(* IEC 61131-3 sources: 2026_Projet_YGO_ExcavatriceDragage/DOC/WFLOW/AUDITS, 1 file *)

(* ---- FB_Cycle_proposal.st ---- *)
(* ═══════════════════════════════════════════════════════════════
   🔄 FB_Cycle — Séquenceur du Cycle Automatique (Grafcet de dragage)
   ───────────────────────────────────────────────────────────────
   📄 Doc : DOC/AF/AF_Partie-04_Mode_SemiAuto_Sequenceur_v2.0.md
            DOC/WFLOW/AUDITS/DESIGN_SEMI_AUTO_CYCLE_v0.1.md
   🔌 Conforme au contrat FB standard (Partie3 §1bis) + §11bis R1-R9.
   🧩 Deux instances : instCycleMaintenance (MAINT_N1/N2) et
      instCycleSemiAuto (SEMI_AUTO) — gating sorties par mode.
   🕹️ Homme-mort (D2) : appui = autorisation 3 s ; mouvement continue
      sans appui ; arrêt au centre du manche (CycleMotionPermit).
   ⏱️ Tempo max d'étape : lancée SEULEMENT si pilotage joystick actif.
   🧊 CycleStepAtError : étape spécifique mémorisée avant STABILIZING (R9).
   🏁 Début de graphe : à la TRÉMIE, treuils en position HAUTE — rebouclage sur X0.
   ═══════════════════════════════════════════════════════════════ *)

FUNCTION_BLOCK PUBLIC FB_Cycle
VAR_INPUT
    Enable                  : BOOL;         // Activation générale du séquenceur
    Reset                   : BOOL;         // Acquittement défaut (front)
    PowerContactorEngaged   : BOOL;         // Chaîne de sécurité OK
    Mode                    : E_Mode;       // Mode arbitré (SEMI_AUTO pour l'instance cycle)
    CycleMotionPermit       : BOOL;         // 🕹️ Manche défléchi (non centré) — D2
    DeadmanArmed            : BOOL;         // 🔫 Appui homme-mort (fenêtre 3 s)
    HeartbeatIhmOk          : BOOL;         // 💓 IHM↔PLC valide

    // Commandes opérateur
    StartCycle              : BOOL;         // Demande lancement / reprise (IHM)
    AbortCycle              : BOOL;         // Demande abandon (IHM) — pas de Pause (D3)

    // Cibles et paramètres (réutilise config maintenance — Q4)
    SelTarget               : INT;          // 🎯 Cible sélectionnée (GVL_IHM.TranslationM3.Cmd.SelTarget) : 1=Trémie, 2=P2, 3=P1, 4=Maintenance
    SetDepthM               : REAL;         // Profondeur de consigne (négative)
    SetOffsetM              : REAL;         // Écart de fermeture benne cible

    // Feedbacks physique & matériel
    KoboldContactFond       : BOOL;         // Retour dédié Kobold : TRUE = contact fond
    LimitLegalReached       : BOOL;         // Limite légale atteinte (descente interdite)
    LimitLegalDepthM        : REAL;         // Profondeur légale minimale autorisée
    WinchSyncError          : BOOL;         // Désynchronisme bloquant M1/M2
    WinchSyncDeltaM         : REAL;         // Écart codeurs M1/M2 pour diagnostic
    M1_CablePosM            : REAL;         // Position câble treuil M1 (recalée)
    M2_CablePosM            : REAL;         // Position câble treuil M2 (recalée)
    M1_MeasuredSpeedMps     : REAL;         // Vitesse linéaire mesurée M1 (m/s)
    M2_MeasuredSpeedMps     : REAL;         // Vitesse linéaire mesurée M2 (m/s)
    SpeedMismatchThresholdMps : REAL;       // Seuil écart vitesse ; 0 = contrôle désactivé
    SpeedMismatchTimeout    : TIME;         // Durée de confirmation ; 0 = contrôle désactivé
    CableLimitM1AscentM     : REAL;         // Limite haute d'exploitation M1

    // Feedbacks Translation M3
    Translation_At_P1           : BOOL;     // Capteur position P1 (arrêt travail)
    Translation_At_Tremie       : BOOL;     // Capteur fin de course trémie
    Translation_At_Maintenance : BOOL;     // Capteur fin de course maintenance
    Translation_Busy            : BOOL;     // Mouvement translation en cours
    Translation_Done            : BOOL;     // Cible translation atteinte

    // Feedbacks Benne
    Benne_Busy              : BOOL;         // Mouvement mâchoires benne en cours
    Benne_Done              : BOOL;         // Mouvement ouverture/fermeture terminé
    Benne_IsOpen            : BOOL;         // Benne mécaniquement ouvert mémorisé
    Benne_IsClosed          : BOOL;         // Benne mécaniquement fermé mémorisé
    Benne_IsRoughlyClosed   : BOOL;         // 🆕 Benne « à peu près fermée » (tolérance matière)

    // 🆕 Référencement (X1_HOMING)
    HomedM1                 : BOOL;         // Codeur M1 référencé
    HomedM2                 : BOOL;         // Codeur M2 référencé
    TopPositionSensor       : BOOL;         // Capteur position haute (référencement)
    HomingRequest           : BOOL;         // Demande de référencement (front)
END_VAR
VAR_OUTPUT
    Ready                   : BOOL;         // Séquenceur disponible
    Busy                    : BOOL;         // Cycle automatique actif
    Done                    : BOOL;         // Cycle automatique complété
    Error                   : BOOL;         // Défaut cycle
    ErrorId                 : WORD;         // bit0: timeout/limite, bit1: désynchronisme, bit2: cible invalide, bit3: stabilisation impossible, bit4: écart vitesse, bit5: perte heartbeat, bit6: tempo max étape
    SpeedMismatchMps        : REAL;         // Écart absolu vitesse M1/M2 (m/s)
    SpeedMismatchActive     : BOOL;         // Seuil vitesse dépassé sur le cycle courant
    SpeedMismatchConfirmed  : BOOL;         // Écart vitesse confirmé pendant SpeedMismatchTimeout

    // Commandes structurées (demandes de mouvement)
    WinchM1Cmd              : ST_WinchCmdDemand;        // Demande treuil M1
    WinchM2Cmd              : ST_WinchCmdDemand;        // Demande treuil M2
    TranslationCmd          : ST_TranslationCmdDemand;  // Demande translation M3
    BucketCmd               : ST_BucketCmdDemand;       // Demande benne

    // Métadonnées d'affichage IHM
    CycleStep               : E_CycleStep;  // Étape active du Grafcet
    CycleStateStr           : STRING(80);   // Libellé en clair de l'étape (Xn - texte)
    CycleStepAtError        : E_CycleStep;  // 🧊 Étape spécifique au moment du défaut (R9)
    SampleCount             : INT;          // 🆕 Compteur de prélèvements (RETAIN, Q3bis)
END_VAR
VAR
    ResetEdge               : R_TRIG;
    StartEdge               : R_TRIG;
    AbortEdge               : R_TRIG;
    ErrorEdge               : R_TRIG;       // 🧊 Capture CycleStepAtError avant bascule (R9)

    // Séquencement
    State                   : E_CycleStep := E_CycleStep.X0_PREPARATION;
    SavedState              : E_CycleStep := E_CycleStep.X0_PREPARATION;

    // Mémorisations et Timers
    TouchPositionM          : REAL;         // Position M1 mémorisée lors du contact fond
    RaiseTargetM            : REAL;         // Profondeur de remontée mémorisée
    DrainingTimer           : TON;          // Temporisateur de vidage (égouttage)
    StabilizationTimer      : TON;          // Temporisation maximale de remontée lente
    SpeedMismatchTimer      : TON;          // Confirmation temporelle écart de vitesse
    StepMaxTimer            : TON;          // 🆕 Tempo max d'étape (R5) — lancée si pilotage
    SelectedWorkTarget      : INT;          // Cible de travail mémorisée (1=Trémie, 3=P1, 4=Maintenance)

    // Paramètres internes
    CtrlAscentDistM         : REAL := 2.0;      // Distance de remontée lente de contrôle
    CtrlAscentToleranceM    : REAL := 0.25;     // Écart maximal admis entre les deux codeurs
    CtrlAscentTimeout       : TIME := T#30s;    // Temps max pour atteindre la zone de stabilisation
    DrainingTime            : TIME := T#5s;     // Temps d'égouttage par défaut
    StepMaxTimeout          : TIME := T#60s;   // 🆕 Tempo max d'étape (à valider, Q4)
END_VAR

// === IMPLEMENTATION ===

{region "Gate securite"}
// 🛑 1. GATES DE SÉCURITÉ ET BLOCAGE (R8)
IF NOT Enable OR NOT PowerContactorEngaged THEN
    WinchM1Cmd.StartStop   := FALSE;
    WinchM1Cmd.Direction   := 0;
    WinchM1Cmd.SpeedPct    := 0.0;

    WinchM2Cmd.StartStop   := FALSE;
    WinchM2Cmd.Direction   := 0;
    WinchM2Cmd.SpeedPct    := 0.0;

    TranslationCmd.Start   := FALSE;
    TranslationCmd.Target  := 0;

    BucketCmd.Open         := FALSE;
    BucketCmd.Close        := FALSE;
    BucketCmd.KoboldContactorCmd := FALSE;

    State                := E_CycleStep.X0_PREPARATION;   // retour à la PREMIÈRE étape (R8)
    CycleStep            := E_CycleStep.X0_PREPARATION;
    CycleStateStr        := 'X0 - Désactivé : sécurité absente ou auto désactivé';
    Ready                := FALSE;
    Busy                 := FALSE;
    Done                 := FALSE;
    RETURN;
END_IF;
{endregion}

{region "Preparation surveillance et commandes cycle"}
Ready := TRUE;
ResetEdge(CLK := Reset);
StartEdge(CLK := StartCycle);
AbortEdge(CLK := AbortCycle);
ErrorEdge(CLK := Error);

// 🧊 R9 — capture l'étape spécifique AVANT la bascule vers STABILIZING
IF ErrorEdge.Q THEN
    CycleStepAtError := State;
END_IF;

// ⏱️ T36 — surveillance indépendante de la remontée lente
StabilizationTimer(IN := (State = E_CycleStep.X7_CTRL_ASCENT), PT := CtrlAscentTimeout);

// 📏 T43 — comparaison vitesse réelle M1/M2
SpeedMismatchMps := ABS(M1_MeasuredSpeedMps - M2_MeasuredSpeedMps);
SpeedMismatchActive := (State = E_CycleStep.X7_CTRL_ASCENT)
                       AND CycleMotionPermit
                       AND (SpeedMismatchThresholdMps > 0.0)
                       AND (SpeedMismatchTimeout > T#0ms)
                       AND (SpeedMismatchMps > SpeedMismatchThresholdMps);
SpeedMismatchTimer(IN := SpeedMismatchActive, PT := SpeedMismatchTimeout);
SpeedMismatchConfirmed := SpeedMismatchTimer.Q;

// 🆕 Tempo max d'étape (R5) — lancée SEULEMENT si pilotage joystick actif (pas de défaut au repos)
StepMaxTimer(IN := CycleMotionPermit AND (State <> E_CycleStep.X0_PREPARATION)
                  AND (State <> E_CycleStep.X13_DONE_SYNC)
                  AND (State <> E_CycleStep.STABILIZING),
             PT := StepMaxTimeout);

IF ResetEdge.Q THEN
    Error := FALSE;
    ErrorId := 16#0000;
    SavedState := E_CycleStep.X0_PREPARATION;
    IF State = E_CycleStep.STABILIZING THEN
        State := E_CycleStep.X0_PREPARATION;
    END_IF;
END_IF;

// 💓 Perte IHM : repli mémorisé. La reconnexion seule ne relance jamais le cycle.
IF NOT HeartbeatIhmOk AND State <> E_CycleStep.STABILIZING THEN
    Error := TRUE;
    ErrorId := ErrorId OR 16#0020;
    State := E_CycleStep.STABILIZING;
END_IF;

// Défaut de synchronisme : arrêt sûr et acquittement obligatoire.
IF WinchSyncError AND State <> E_CycleStep.STABILIZING THEN
    Error := TRUE;
    ErrorId := ErrorId OR 16#0002;
    State := E_CycleStep.STABILIZING;
END_IF;

// 🛡️ T43 — écart de vitesse confirmé : arrêt du cycle et STABILIZING.
IF SpeedMismatchConfirmed AND State <> E_CycleStep.STABILIZING THEN
    Error := TRUE;
    ErrorId := ErrorId OR 16#0010;
    State := E_CycleStep.STABILIZING;
END_IF;

// 🆕 Tempo max d'étape dépassée (blocage probable) → défaut
IF StepMaxTimer.Q AND State <> E_CycleStep.STABILIZING THEN
    Error := TRUE;
    ErrorId := ErrorId OR 16#0040;
    State := E_CycleStep.STABILIZING;
END_IF;

// Gestion de l'Abandon (D3 — pas de Pause)
IF AbortEdge.Q THEN
    State := E_CycleStep.X0_PREPARATION;
END_IF;
{endregion}

{region "Machine etat cycle automatique"}
// 🔁 2. LOGIQUE DU SÉQUENCEUR (Machine d'état) — CASE sur enum unique (R1)
CASE State OF

    E_CycleStep.X0_PREPARATION:
        CycleStep := E_CycleStep.X0_PREPARATION;
        CycleStateStr := 'X0 - Vérification cohérence système';
        WinchM1Cmd.StartStop := FALSE; WinchM1Cmd.Direction := 0; WinchM1Cmd.SpeedPct := 0.0;
        WinchM2Cmd.StartStop := FALSE; WinchM2Cmd.Direction := 0; WinchM2Cmd.SpeedPct := 0.0;
        TranslationCmd.Start := FALSE; TranslationCmd.Target := 0;
        BucketCmd.Open := FALSE; BucketCmd.Close := FALSE; BucketCmd.KoboldContactorCmd := FALSE;
        Busy := FALSE; Done := FALSE;

        // Transition si système sain et réarmé (front reset ou démarrage)
        IF StartEdge.Q THEN
            State := E_CycleStep.X1_HOMING;
        END_IF;

    E_CycleStep.X1_HOMING:
        CycleStep := E_CycleStep.X1_HOMING;
        CycleStateStr := 'X1 - Référencement codeurs (vitesses lentes)';
        Busy := TRUE;

        // 🆕 Vitesses lentes pour chercher capteur top + référencement
        IF NOT HomedM1 OR NOT HomedM2 THEN
            WinchM1Cmd.StartStop := CycleMotionPermit;
            WinchM1Cmd.Direction := 1;   // montée lente vers capteur top
            WinchM1Cmd.SpeedPct := 10.0;
            WinchM2Cmd.StartStop := CycleMotionPermit;
            WinchM2Cmd.Direction := 1;
            WinchM2Cmd.SpeedPct := 10.0;
            IF HomingRequest THEN
                // déclenche le référencement (via FB_Encoder_Homing en aval)
                State := E_CycleStep.X2_WORK_POS_SELECT;
            END_IF;
        ELSE
            // déjà homé → passe vite
            State := E_CycleStep.X2_WORK_POS_SELECT;
        END_IF;

    E_CycleStep.X2_WORK_POS_SELECT:
        CycleStep := E_CycleStep.X2_WORK_POS_SELECT;
        CycleStateStr := 'X2 - Sélection position travail (P1)';
        Busy := TRUE;

        // 🆕 Destinations sélectionnables : Trémie(1), P1(3), Maintenance(4).
        // P2(2) n'est PAS une destination — capteur de passage en petite vitesse (PV).
        IF (SelTarget <> 1) AND (SelTarget <> 3) AND (SelTarget <> 4) THEN
            Error := TRUE;
            ErrorId := ErrorId OR 16#0004;
            State := E_CycleStep.STABILIZING;
        ELSE
            SelectedWorkTarget := SelTarget;
            TranslationCmd.Target := SelTarget;
            TranslationCmd.Start := CycleMotionPermit;
            // Arrivée à la cible (Trémie/P1/Maintenance) — capteurs PV/PVP2/P2 = ralentissement
            IF CycleMotionPermit AND (
                (SelTarget = 1 AND Translation_At_Tremie) OR
                (SelTarget = 3 AND Translation_At_P1) OR
                (SelTarget = 4 AND Translation_At_Maintenance)) THEN
                TranslationCmd.Start := FALSE;
                State := E_CycleStep.X3_OPEN_BUCKET;
            END_IF;
        END_IF;

    E_CycleStep.X3_OPEN_BUCKET:
        CycleStep := E_CycleStep.X3_OPEN_BUCKET;
        CycleStateStr := 'X3 - Ouverture benne';
        Busy := TRUE;

        // 🆕 Ouverture benne ; si déjà ouverte → passe vite
        IF Benne_IsOpen THEN
            State := E_CycleStep.X4_DESCEND_OPEN;
        ELSE
            BucketCmd.Open := CycleMotionPermit;
            IF CycleMotionPermit AND Benne_Done AND Benne_IsOpen THEN
                BucketCmd.Open := FALSE;
                State := E_CycleStep.X4_DESCEND_OPEN;
            END_IF;
        END_IF;

    E_CycleStep.X4_DESCEND_OPEN:
        CycleStep := E_CycleStep.X4_DESCEND_OPEN;
        CycleStateStr := 'X4 - Plongée benne ouverte (synchro)';

        // M1 et M2 descendent ensemble (synchro gérée en aval)
        WinchM1Cmd.StartStop := CycleMotionPermit;
        WinchM1Cmd.Direction := -1;
        WinchM1Cmd.SpeedPct  := 50.0;
        WinchM2Cmd.StartStop := CycleMotionPermit;
        WinchM2Cmd.Direction := -1;
        WinchM2Cmd.SpeedPct  := 50.0;
        BucketCmd.KoboldContactorCmd := TRUE;

        // Transition uniquement sur le retour dédié Kobold.
        IF CycleMotionPermit AND KoboldContactFond THEN
            WinchM1Cmd.StartStop := FALSE;
            WinchM2Cmd.StartStop := FALSE;
            BucketCmd.KoboldContactorCmd := FALSE;
            TouchPositionM := M1_CablePosM;
            IF LimitLegalDepthM < -0.01 THEN
                RaiseTargetM := MAX(TouchPositionM + 0.5, LimitLegalDepthM + 0.5);
            ELSE
                RaiseTargetM := TouchPositionM + 0.5;
            END_IF;
            State := E_CycleStep.X5_BOTTOM_CONFIRMED;
        ELSIF LimitLegalReached THEN
            Error := TRUE;
            ErrorId := ErrorId OR 16#0001;
            WinchM1Cmd.StartStop := FALSE;
            WinchM2Cmd.StartStop := FALSE;
            BucketCmd.KoboldContactorCmd := FALSE;
            State := E_CycleStep.STABILIZING;
        END_IF;

    E_CycleStep.X5_BOTTOM_CONFIRMED:
        CycleStep := E_CycleStep.X5_BOTTOM_CONFIRMED;
        CycleStateStr := 'X5 - Fond confirmé : remontée sécurisée';

        WinchM1Cmd.StartStop := CycleMotionPermit;
        WinchM1Cmd.Direction := 1;
        WinchM1Cmd.SpeedPct := 20.0;
        WinchM2Cmd.StartStop := CycleMotionPermit;
        WinchM2Cmd.Direction := 1;
        WinchM2Cmd.SpeedPct := 20.0;

        // Les deux treuils restent synchronisés jusqu'au-dessus de la limite légale.
        IF CycleMotionPermit AND (M1_CablePosM >= RaiseTargetM) AND (M2_CablePosM >= RaiseTargetM) THEN
            WinchM1Cmd.StartStop := FALSE;
            WinchM2Cmd.StartStop := FALSE;
            State := E_CycleStep.X6_CLOSE_BUCKET;
        END_IF;

    E_CycleStep.X6_CLOSE_BUCKET:
        CycleStep := E_CycleStep.X6_CLOSE_BUCKET;
        CycleStateStr := 'X6 - Fermeture benne (tolérance à peu près fermé)';

        WinchM1Cmd.StartStop := FALSE;
        BucketCmd.Close := TRUE;

        // 🆕 Tolérance : si benne « à peu près fermée » (matière/objet), on remonte et on contrôle
        IF CycleMotionPermit AND (Benne_Done AND (Benne_IsClosed OR Benne_IsRoughlyClosed)) THEN
            BucketCmd.Close := FALSE;
            State := E_CycleStep.X7_CTRL_ASCENT;
        END_IF;

    E_CycleStep.X7_CTRL_ASCENT:
        CycleStep := E_CycleStep.X7_CTRL_ASCENT;
        CycleStateStr := 'X7 - Remontée lente de contrôle';

        WinchM1Cmd.StartStop := CycleMotionPermit;
        WinchM1Cmd.Direction := 1;
        WinchM1Cmd.SpeedPct  := 20.0;
        WinchM2Cmd.StartStop := CycleMotionPermit;
        WinchM2Cmd.Direction := 1;
        WinchM2Cmd.SpeedPct  := 20.0;

        // Contrôle des deux codeurs
        IF WinchSyncError OR (ABS(M1_CablePosM - M2_CablePosM) > CtrlAscentToleranceM) THEN
            Error := TRUE;
            ErrorId := ErrorId OR 16#0008;
            State := E_CycleStep.STABILIZING;
        ELSIF CycleMotionPermit
           AND (M1_CablePosM >= (TouchPositionM + CtrlAscentDistM))
           AND (M2_CablePosM >= (TouchPositionM + CtrlAscentDistM))
           AND (ABS(M1_CablePosM - M2_CablePosM) <= CtrlAscentToleranceM) THEN
            State := E_CycleStep.X8_ASCENT_LOADED;
        ELSIF StabilizationTimer.Q THEN
            Error := TRUE;
            ErrorId := ErrorId OR 16#0008;
            State := E_CycleStep.STABILIZING;
        END_IF;

    E_CycleStep.X8_ASCENT_LOADED:
        CycleStep := E_CycleStep.X8_ASCENT_LOADED;
        CycleStateStr := 'X8 - Remontée en charge';

        WinchM1Cmd.StartStop := CycleMotionPermit;
        WinchM1Cmd.Direction := 1;
        WinchM1Cmd.SpeedPct  := 70.0;
        WinchM2Cmd.StartStop := CycleMotionPermit;
        WinchM2Cmd.Direction := 1;
        WinchM2Cmd.SpeedPct  := 70.0;

        // Transition alignée sur la limite haute d'exploitation
        IF CycleMotionPermit AND M1_CablePosM >= CableLimitM1AscentM THEN
            WinchM1Cmd.StartStop := FALSE;
            WinchM2Cmd.StartStop := FALSE;
            State := E_CycleStep.X9_DRAIN_PAUSE;
        END_IF;

    E_CycleStep.X9_DRAIN_PAUSE:
        CycleStep := E_CycleStep.X9_DRAIN_PAUSE;
        CycleStateStr := 'X9 - Égouttage du godet en cours';
        WinchM1Cmd.StartStop := FALSE;
        WinchM2Cmd.StartStop := FALSE;

        DrainingTimer(IN := TRUE, PT := DrainingTime);
        // 🆕 Temps écoulé affiché IHM (CycleStateStr + champ dédié)
        IF CycleMotionPermit AND DrainingTimer.Q THEN
            DrainingTimer(IN := FALSE);
            State := E_CycleStep.X10_TRANSLATE_DUMP;
        END_IF;

    E_CycleStep.X10_TRANSLATE_DUMP:
        CycleStep := E_CycleStep.X10_TRANSLATE_DUMP;
        CycleStateStr := 'X10 - Déplacement vers trémie (grille/crible libres)';

        TranslationCmd.Target := 1; // Trémie
        TranslationCmd.Start := CycleMotionPermit;

        // 🆕 Avertissement IHM : grille abaissée/libre, crible libre pour réceptionner la charge
        // (porté par CycleStateStr + OperatorAction côté supervision)

        // Transition si translation arrivé à la trémie
        IF CycleMotionPermit AND Translation_At_Tremie THEN
            TranslationCmd.Start := FALSE;
            State := E_CycleStep.X11_OPEN_DUMP;
        END_IF;

    E_CycleStep.X11_OPEN_DUMP:
        CycleStep := E_CycleStep.X11_OPEN_DUMP;
        CycleStateStr := 'X11 - Vidange / ouverture du godet (montée possible, descente ouvre)';

        // 🆕 Montée possible (treuils vers le haut) ; descente fait ouvrir la benne.
        // Montée : on laisse l'opérateur remonter les 2 treuils en synchro si besoin.
        WinchM1Cmd.StartStop := CycleMotionPermit AND (WinchM1Cmd.Direction = 1);
        WinchM1Cmd.Direction := 1;
        WinchM1Cmd.SpeedPct  := 20.0;
        WinchM2Cmd.StartStop := CycleMotionPermit AND (WinchM2Cmd.Direction = 1);
        WinchM2Cmd.Direction := 1;
        WinchM2Cmd.SpeedPct  := 20.0;

        // Descente → ouverture benne (vidage)
        BucketCmd.Open := CycleMotionPermit AND (WinchM1Cmd.Direction = -1);

        // 🆕 Contrôle convoyeurs par MESSAGE utilisateur (pas encore câblé) :
        // CycleStateStr + OperatorAction côté supervision demandent de vérifier
        // que les convoyeurs sont en route avant/au lâcher.
        IF CycleMotionPermit AND Benne_Done AND Benne_IsOpen THEN
            BucketCmd.Open := FALSE;
            State := E_CycleStep.X13_DONE_SYNC;
        END_IF;

    E_CycleStep.X13_DONE_SYNC:
        CycleStep := E_CycleStep.X13_DONE_SYNC;
        CycleStateStr := 'X13 - Cycle automatique complété - prêt';
        WinchM1Cmd.StartStop := FALSE;
        WinchM2Cmd.StartStop := FALSE;
        TranslationCmd.Start := FALSE;
        Done := TRUE;
        Busy := FALSE;

        // 🆕 Compteur de prélèvements (RETAIN, Q3bis) — compte inconditionnellement
        SampleCount := SampleCount + 1;

        // 🆕 Rebouclage sur X0_PREPARATION (trémie, treuils hauts) — pas de retour P1
        IF StartEdge.Q THEN
            Done := FALSE;
            State := E_CycleStep.X0_PREPARATION;
        END_IF;

    E_CycleStep.STABILIZING:
        CycleStep := E_CycleStep.STABILIZING;
        CycleStateStr := 'X14 - Cycle en attente / stabilisation (STAB)';
        WinchM1Cmd.StartStop := FALSE;
        WinchM2Cmd.StartStop := FALSE;
        TranslationCmd.Start := FALSE;
        BucketCmd.Open := FALSE;
        BucketCmd.Close := FALSE;

END_CASE;
{endregion}

{region "Repli homme mort"}
// 🛑 Relâchement du manche (retour au centre) : aucune demande d'actionneur ne reste active.
// L'étape est mémorisée et reprend au prochain appui valide (D2).
IF Busy AND NOT CycleMotionPermit THEN
    WinchM1Cmd.StartStop := FALSE;
    WinchM2Cmd.StartStop := FALSE;
    TranslationCmd.Start := FALSE;
    BucketCmd.Open := FALSE;
    BucketCmd.Close := FALSE;
    BucketCmd.KoboldContactorCmd := FALSE;
END_IF;
{endregion}

END_FUNCTION_BLOCK
